// TIA Portal project "the last one" (V15)

(* hardware
DEVICE "S7-1200 station_1"  S7-1200 Station
   slot 0: "Rack_0"  S7-1200 Rack  Rack  V1.0
   slot 1: "PLC_1"  CPU 1212C AC/DC/Rly  6ES7 212-1BE40-0XB0  V4.0
   slot 101: "CM 1241 (RS422/485)_1"  6ES7 241-1CH32-0XB0  V2.2
DEVICE "S7-1200 station_3"  S7-1200 Station
   slot 0: "Rack_0"  S7-1200 Rack  Rack  V1.0
   slot 1: "PLC_3"  CPU 1212C AC/DC/Rly  6ES7 212-1BE31-0XB0  V3.0
*)

// ===== PLC "PLC_1"  CPU 1212C AC/DC/Rly =====

VAR_GLOBAL   // PLC tag table "Default tag table"
   "System_Byte" AT %MB1 : Byte;
   "FirstScan" AT %M1.0 : Bool;
   "DiagStatusUpdate" AT %M1.1 : Bool;
   "AlwaysTRUE" AT %M1.2 : Bool;
   "AlwaysFALSE" AT %M1.3 : Bool;
   "Clock_Byte" AT %MB0 : Byte;
   "Clock_10Hz" AT %M0.0 : Bool;
   "Clock_5Hz" AT %M0.1 : Bool;
   "Clock_2.5Hz" AT %M0.2 : Bool;
   "Clock_2Hz" AT %M0.3 : Bool;
   "Clock_1.25Hz" AT %M0.4 : Bool;
   "Clock_1Hz" AT %M0.5 : Bool;
   "Clock_0.625Hz" AT %M0.6 : Bool;
   "Clock_0.5Hz" AT %M0.7 : Bool;
   "Tag_1" AT %M2.0 : Bool;
   "Tag_2" AT %M2.1 : Bool;
   "Tag_3" AT %M2.2 : Bool;
   "Tag_4" AT %M2.3 : Bool;
   "Tag_5" AT %M2.4 : Bool;
   "Tag_6" AT %M2.5 : Bool;
   "freq" AT %MW10 : Word;
   "run" AT %MW12 : Word;
   "freq.refrance" AT %MW14 : Word;
   "volt" AT %MW16 : Word;
   "current" AT %MW18 : Word;
   "atomatic" AT %M2.6 : Bool;
   "manual" AT %M2.7 : Bool;
   "incoder_input" AT %ID1000 : DWord;
   "encoder" AT %MD40 : DInt;
   "panda(1)" AT %M3.0 : Bool;
   "start" AT %I0.1 : Bool;
   "reset" AT %I0.2 : Bool;
   "stop" AT %I0.3 : Bool;
   "stop_scada" AT %M3.1 : Bool;
   "reset_scada" AT %M3.2 : Bool;
   "start_scada" AT %M3.4 : Bool;
   "Tag_7" AT %M3.5 : Bool;
   "Tag_8" AT %M3.6 : Bool;
   "red" AT %MW20 : Word;
   "Tag_9" AT %MW22 : Int;
   "Tag_10" AT %M3.7 : Bool;
   "red valve" AT %Q0.0 : Bool;
   "Tag_11" AT %M4.0 : Bool;
   "Tag_12" AT %MW100 : Int;
   "Tag_13" AT %M4.1 : Bool;
   "Tag_14" AT %M4.2 : Bool;
   "reverse" AT %M4.3 : Bool;
   "Tag_15" AT %M4.4 : Bool;
   "Tag_16" AT %M4.5 : Bool;
   "Tag_17" AT %M4.6 : Bool;
   "Tag_18" AT %M4.7 : Bool;
   "green" AT %MW24 : Int;
   "Tag_19" AT %MW26 : Int;
   "green valve" AT %Q0.1 : Bool;
   "Tag_20" AT %M5.0 : Bool;
   "Tag_21" AT %M5.1 : Bool;
   "Tag_22" AT %M5.2 : Bool;
   "Tag_23" AT %M5.3 : Bool;
   "Tag_24" AT %M5.4 : Bool;
   "Tag_25" AT %M5.5 : Bool;
   "blue" AT %MW28 : Int;
   "Tag_27" AT %MW30 : Int;
   "blue valve" AT %Q0.2 : Bool;
   "Tag_28" AT %M5.6 : Bool;
   "Tag_26" AT %M5.7 : Bool;
   "Tag_29" AT %M6.0 : Bool;
   "Tag_30" AT %M6.1 : Bool;
   "Tag_31" AT %M6.2 : Bool;
   "Tag_32" AT %M6.3 : Bool;
   "Tag_33" AT %M6.4 : Bool;
   "Tag_34" AT %M6.5 : Bool;
   "Tag_35" AT %M6.6 : Bool;
   "Tag_36" AT %M6.7 : Bool;
   "cylinder" AT %Q0.3 : Bool;
   "Tag_37" AT %M7.0 : Bool;
   "mixer" AT %Q0.4 : Bool;
   "forward" AT %M7.1 : Bool;
   "Tag_38" AT %M7.2 : Bool;
   "Tag_39" AT %M7.3 : Bool;
   "Tag_40" AT %M7.5 : Bool;
   "Tag_41" AT %M7.6 : Bool;
   "Tag_42" AT %M7.7 : Bool;
   "Tag_43" AT %M8.0 : Bool;
   "Tag_44" AT %M8.1 : Bool;
   "Tag_45" AT %M8.2 : Bool;
   "m_redvalve" AT %M8.3 : Bool;
   "m_greenvalve" AT %M8.4 : Bool;
   "Tag_48" AT %M8.5 : Bool;
   "m_bluevalve" AT %M8.6 : Bool;
   "m_forward" AT %M8.7 : Bool;
   "m_reverse" AT %M9.0 : Bool;
   "Tag_52" AT %M9.1 : Bool;
   "Tag_46" AT %M9.2 : Bool;
   "Tag_47" AT %M9.3 : Bool;
   "Tag_49" AT %M9.4 : Bool;
   "Tag_50" AT %M34.0 : Bool;
   "Tag_51" AT %M90.0 : Bool;
   "Tag_53" AT %MW102 : Int;
   "Tag_54" AT %MW104 : Int;
   "Tag_55" AT %M90.1 : Bool;
   "Tag_56" AT %MD50 : DWord;
   "Tag_57" AT %MD54 : DWord;
   "Tag_58" AT %M50.0 : Bool;
   "Tag_59" AT %M50.1 : Bool;
   "n0" AT %M58.0 : Bool;
   "n1" AT %M58.1 : Bool;
   "n2" AT %M58.2 : Bool;
   "n3" AT %M58.3 : Bool;
   "n4" AT %M58.4 : Bool;
   "n5" AT %M58.5 : Bool;
   "n6" AT %M58.6 : Bool;
   "n7" AT %M58.7 : Bool;
   "p0" AT %M59.0 : Bool;
   "p1" AT %M59.1 : Bool;
   "p2" AT %M59.2 : Bool;
   "p3" AT %M59.3 : Bool;
   "p4" AT %M59.4 : Bool;
   "p5" AT %M59.5 : Bool;
   "p6" AT %M59.6 : Bool;
   "p7" AT %M59.7 : Bool;
   "p8" AT %M60.0 : Bool;
   "p9" AT %M60.1 : Bool;
   "X" AT %M110.0 : Bool;
   "Tag_60" AT %MW60 : Int;
   "r0" AT %M62.0 : Bool;
   "r1" AT %M62.1 : Bool;
   "r2" AT %M62.2 : Bool;
   "r3" AT %M62.3 : Bool;
   "r4" AT %M62.4 : Bool;
   "r5" AT %M62.5 : Bool;
   "r6" AT %M62.6 : Bool;
   "r7" AT %M62.7 : Bool;
   "r8" AT %M63.0 : Bool;
   "r9" AT %M63.1 : Bool;
   "t1" AT %M63.2 : Bool;
   "t2" AT %M63.3 : Bool;
   "t3" AT %M63.4 : Bool;
   "t4" AT %M63.5 : Bool;
   "t5" AT %M63.6 : Bool;
   "t6" AT %M63.7 : Bool;
   "t7" AT %M64.0 : Bool;
   "t8" AT %M64.1 : Bool;
   "Tag_61" AT %MW80 : Int;
   "Tag_62" AT %MW120 : Word;
   "Tag_63" AT %MW90 : Int;
   "Tag_64" AT %MW40 : Word;
   "Tag_65" AT %MW82 : Int;
   "Tag_66" AT %MW122 : Word;
   "Tag_67" AT %MW92 : Int;
   "Tag_68" AT %MW124 : Word;
   "Tag_69" AT %MW94 : Int;
   "Tag_70" AT %MW84 : Int;
   "Tag_71" AT %MW130 : Int;
   "Tag_72" AT %MW132 : Int;
   "Tag_73" AT %MW134 : Int;
   "Tag_74" AT %MW136 : Int;
   "p11" AT %M138.0 : Bool;
   "p12" AT %M138.1 : Bool;
   "p13" AT %M138.2 : Bool;
   "p14" AT %M138.3 : Bool;
   "Tag_75" AT %MW50 : Word;
   "rstop" AT %M138.4 : Bool;
   "Tag_76" AT %MW86 : Word;
   "Tag_77" AT %M87.0 : Bool;
   "Tag_78" AT %M87.1 : Bool;
   "Tag_79" AT %M87.5 : Bool;
   "Tag_80" AT %M150.0 : Bool;
   "Tag_81" AT %M150.2 : Bool;
   "Tag_82" AT %M150.3 : Bool;
   "Tag_83" AT %M150.4 : Bool;
   "Tag_84" AT %M150.5 : Bool;
   "Tag_85" AT %M150.6 : Bool;
   "Tag_86" AT %M151.0 : Bool;
   "Tag_87" AT %M151.2 : Bool;
   "Tag_88" AT %M153.0 : Bool;
   "valve 1" AT %M160.0 : Bool;
   "valve 2" AT %M160.1 : Bool;
   "valve 3" AT %M160.2 : Bool;
   "cylinder_scada" AT %M160.3 : Bool;
   "mixer_scada" AT %M160.4 : Bool;
   "forward_scada" AT %M160.5 : Bool;
   "reverse_scada" AT %M160.6 : Bool;
   "Tag_89" AT %M166.0 : Bool;
   "Tag_90" AT %M166.1 : Bool;
   "Tag_91" AT %M166.2 : Bool;
   "Tag_92" AT %M166.3 : Bool;
   "Tag_93" AT %M170.0 : Bool;
   "Tag_94" AT %M171.0 : Bool;
   "Tag_95" AT %M170.1 : Bool;
   "Tag_96" AT %M171.1 : Bool;
   "Tag_97" AT %M170.3 : Bool;
   "Tag_98" AT %M171.3 : Bool;
   "Tag_99" AT %M170.2 : Bool;
   "Tag_100" AT %M171.2 : Bool;
END_VAR

DATA_BLOCK "auto_DB"   // DB11
{ S7_Optimized_Access := 'TRUE' }
VERSION : 0.1
// stored: InstanceOfName auto
"auto"
BEGIN
END_DATA_BLOCK

// folder: System blocks/Program resources

DATA_BLOCK "IEC_Counter_0_DB"   // DB4
{ S7_Optimized_Access := 'TRUE' }
AUTHOR : Simatic
FAMILY : IEC
NAME : CNTR
VERSION : 1.0
// stored: InstanceOfName IEC_COUNTER
"IEC_COUNTER"
BEGIN
END_DATA_BLOCK

DATA_BLOCK "IEC_Timer_0_DB"   // DB5
{ S7_Optimized_Access := 'TRUE' }
AUTHOR : Simatic
FAMILY : IEC
NAME : IEC_TMR
VERSION : 1.0
// stored: InstanceOfName IEC_TIMER
"IEC_TIMER"
BEGIN
END_DATA_BLOCK

DATA_BLOCK "IEC_Timer_0_DB_1"   // DB6
{ S7_Optimized_Access := 'TRUE' }
AUTHOR : Simatic
FAMILY : IEC
NAME : IEC_TMR
VERSION : 1.0
// stored: InstanceOfName IEC_TIMER
"IEC_TIMER"
BEGIN
END_DATA_BLOCK

DATA_BLOCK "IEC_Timer_0_DB_2"   // DB7
{ S7_Optimized_Access := 'TRUE' }
AUTHOR : Simatic
FAMILY : IEC
NAME : IEC_TMR
VERSION : 1.0
// stored: InstanceOfName IEC_TIMER
"IEC_TIMER"
BEGIN
END_DATA_BLOCK

DATA_BLOCK "IEC_Timer_0_DB_3"   // DB8
{ S7_Optimized_Access := 'TRUE' }
AUTHOR : Simatic
FAMILY : IEC
NAME : IEC_TMR
VERSION : 1.0
// stored: InstanceOfName IEC_TIMER
"IEC_TIMER"
BEGIN
END_DATA_BLOCK

DATA_BLOCK "IEC_Counter_0_DB_1"   // DB9
{ S7_Optimized_Access := 'TRUE' }
AUTHOR : Simatic
FAMILY : IEC
NAME : CNTR
VERSION : 1.0
// stored: InstanceOfName IEC_COUNTER
"IEC_COUNTER"
BEGIN
END_DATA_BLOCK

DATA_BLOCK "IEC_Timer_0_DB_4"   // DB10
{ S7_Optimized_Access := 'TRUE' }
AUTHOR : Simatic
FAMILY : IEC
NAME : IEC_TMR
VERSION : 1.0
// stored: InstanceOfName IEC_TIMER
"IEC_TIMER"
BEGIN
END_DATA_BLOCK

DATA_BLOCK "IEC_Counter_0_DB_2"   // DB13
{ S7_Optimized_Access := 'TRUE' }
AUTHOR : Simatic
FAMILY : IEC
NAME : CNTR
VERSION : 1.0
// stored: InstanceOfName IEC_COUNTER
"IEC_COUNTER"
BEGIN
END_DATA_BLOCK

DATA_BLOCK "IEC_Counter_0_DB_3"   // DB14
{ S7_Optimized_Access := 'TRUE' }
AUTHOR : Simatic
FAMILY : IEC
NAME : CNTR
VERSION : 1.0
// stored: InstanceOfName IEC_COUNTER
"IEC_COUNTER"
BEGIN
END_DATA_BLOCK

// folder: (top level)

FUNCTION_BLOCK "auto"   // FB1, LAD
{ S7_Optimized_Access := 'TRUE' }
VERSION : 0.1
   VAR_TEMP   // added for the SCL form of the ladder/FBD networks
      _w1 : Bool;
      _w2 : Bool;
      _w3 : Bool;
      _w4 : Bool;
   END_VAR
BEGIN

REGION Network 1
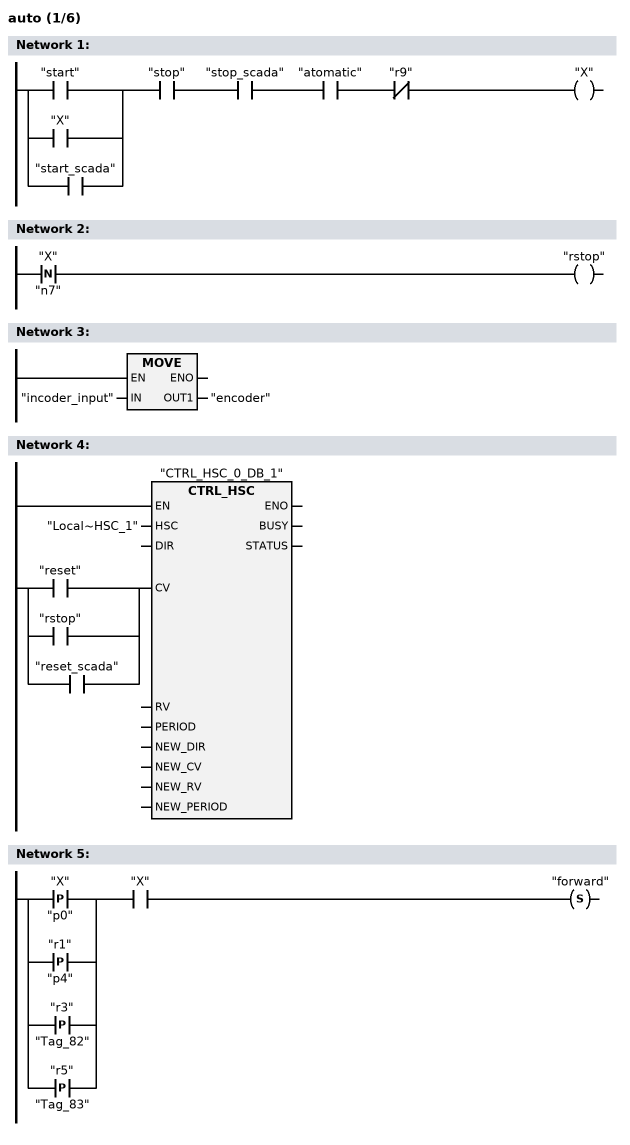
   RUNG wire#powerrail
      Contact( "start" )
      wire#w1
      Contact( "stop" )
      Contact( "stop_scada" )
      Contact( "atomatic" )
      I_Contact( "r9" )
      Coil( "X" )
   END_RUNG
   RUNG wire#powerrail
      Contact( "X" )
   END_RUNG wire#w1
   RUNG wire#powerrail
      Contact( "start_scada" )
   END_RUNG wire#w1
   // the same network as SCL:
   "X" := ("start" OR "X" OR "start_scada") AND "stop" AND "stop_scada" AND "atomatic" AND NOT "r9";
END_REGION

REGION Network 2
   RUNG wire#powerrail
      N_Contact(operand := "X", bit := "n7")
      Coil( "rstop" )
   END_RUNG
   // the same network as SCL:
   #_w1 := NOT "X" AND "n7";   // falling edge of "X"
   "n7" := "X";
   "rstop" := #_w1;
END_REGION

REGION Network 3
   RUNG wire#powerrail
      Move(in := "incoder_input", out1 => "encoder")
   END_RUNG
   // the same network as SCL:
   "encoder" := "incoder_input";
END_REGION

REGION Network 4
   "CTRL_HSC_0_DB_1"(HSC := "Local~HSC_1", CV := "reset" OR "rstop" OR "reset_scada");   // CTRL_HSC
END_REGION

REGION Network 5
   RUNG wire#powerrail
      P_Contact(operand := "X", bit := "p0")
      wire#w1
      Contact( "X" )
      S_Coil( "forward" )
   END_RUNG
   RUNG wire#powerrail
      P_Contact(operand := "r1", bit := "p4")
   END_RUNG wire#w1
   RUNG wire#powerrail
      P_Contact(operand := "r3", bit := "Tag_82")
   END_RUNG wire#w1
   RUNG wire#powerrail
      P_Contact(operand := "r5", bit := "Tag_83")
   END_RUNG wire#w1
   // the same network as SCL:
   #_w1 := "X" AND NOT "p0";   // rising edge of "X"
   "p0" := "X";
   #_w2 := "r1" AND NOT "p4";   // rising edge of "r1"
   "p4" := "r1";
   #_w3 := "r3" AND NOT "Tag_82";   // rising edge of "r3"
   "Tag_82" := "r3";
   #_w4 := "r5" AND NOT "Tag_83";   // rising edge of "r5"
   "Tag_83" := "r5";
   IF (#_w1 OR #_w2 OR #_w3 OR #_w4) AND "X" THEN "forward" := TRUE; END_IF;
END_REGION

REGION Network 6
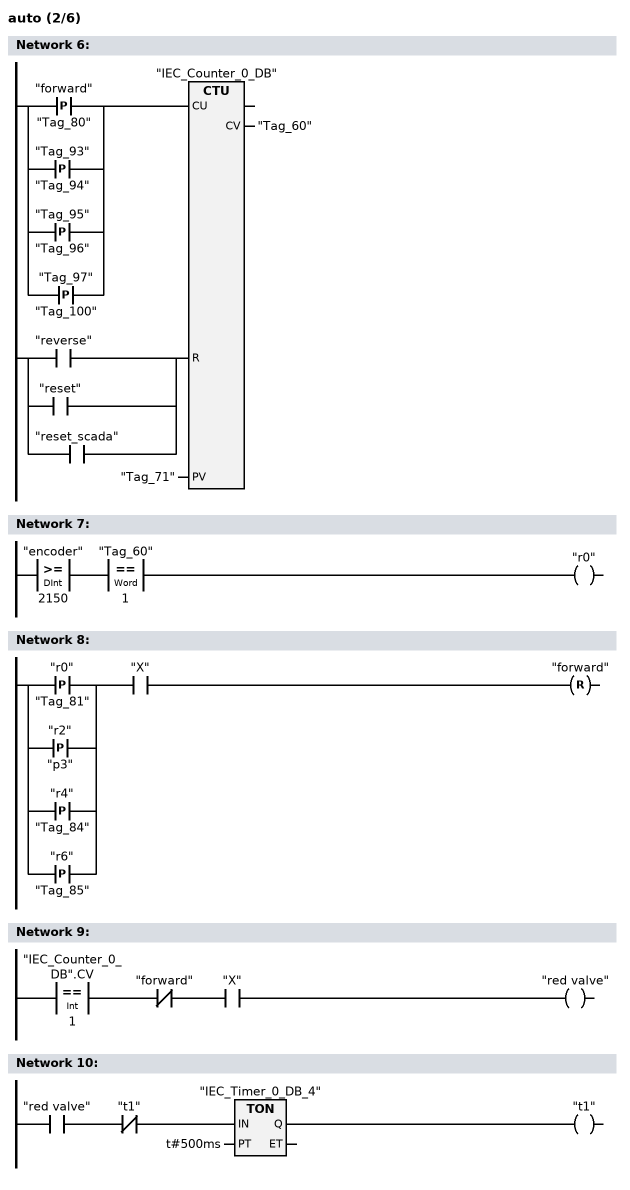
   #_w1 := "forward" AND NOT "Tag_80";   // rising edge of "forward"
   "Tag_80" := "forward";
   #_w2 := "Tag_93" AND NOT "Tag_94";   // rising edge of "Tag_93"
   "Tag_94" := "Tag_93";
   #_w3 := "Tag_95" AND NOT "Tag_96";   // rising edge of "Tag_95"
   "Tag_96" := "Tag_95";
   #_w4 := "Tag_97" AND NOT "Tag_100";   // rising edge of "Tag_97"
   "Tag_100" := "Tag_97";
   "IEC_Counter_0_DB".CTU(CU := #_w1 OR #_w2 OR #_w3 OR #_w4,
                          R := "reverse" OR "reset" OR "reset_scada",
                          PV := "Tag_71",
                          CV => "Tag_60");
END_REGION

REGION Network 7
   RUNG wire#powerrail
      { S7_Templates := "SrcType := DInt" } GE_Contact(in1 := "encoder", in2 := 2150)
      { S7_Templates := "SrcType := Word" } EQ_Contact(in1 := "Tag_60", in2 := 1)
      Coil( "r0" )
   END_RUNG
   // the same network as SCL:
   "r0" := ("encoder" >= 2150) AND ("Tag_60" = 1);
END_REGION

REGION Network 8
   RUNG wire#powerrail
      P_Contact(operand := "r0", bit := "Tag_81")
      wire#w1
      Contact( "X" )
      R_Coil( "forward" )
   END_RUNG
   RUNG wire#powerrail
      P_Contact(operand := "r2", bit := "p3")
   END_RUNG wire#w1
   RUNG wire#powerrail
      P_Contact(operand := "r4", bit := "Tag_84")
   END_RUNG wire#w1
   RUNG wire#powerrail
      P_Contact(operand := "r6", bit := "Tag_85")
   END_RUNG wire#w1
   // the same network as SCL:
   #_w1 := "r0" AND NOT "Tag_81";   // rising edge of "r0"
   "Tag_81" := "r0";
   #_w2 := "r2" AND NOT "p3";   // rising edge of "r2"
   "p3" := "r2";
   #_w3 := "r4" AND NOT "Tag_84";   // rising edge of "r4"
   "Tag_84" := "r4";
   #_w4 := "r6" AND NOT "Tag_85";   // rising edge of "r6"
   "Tag_85" := "r6";
   IF (#_w1 OR #_w2 OR #_w3 OR #_w4) AND "X" THEN "forward" := FALSE; END_IF;
END_REGION

REGION Network 9
   RUNG wire#powerrail
      { S7_Templates := "SrcType := Int" } EQ_Contact(in1 := "IEC_Counter_0_DB".CV, in2 := 1)
      I_Contact( "forward" )
      Contact( "X" )
      Coil( "red valve" )
   END_RUNG
   // the same network as SCL:
   "red valve" := ("IEC_Counter_0_DB".CV = 1) AND NOT "forward" AND "X";
END_REGION

REGION Network 10
   "IEC_Timer_0_DB_4".TON(IN := "red valve" AND NOT "t1", PT := t#500ms);
   "t1" := "IEC_Timer_0_DB_4".Q;
END_REGION

REGION Network 11
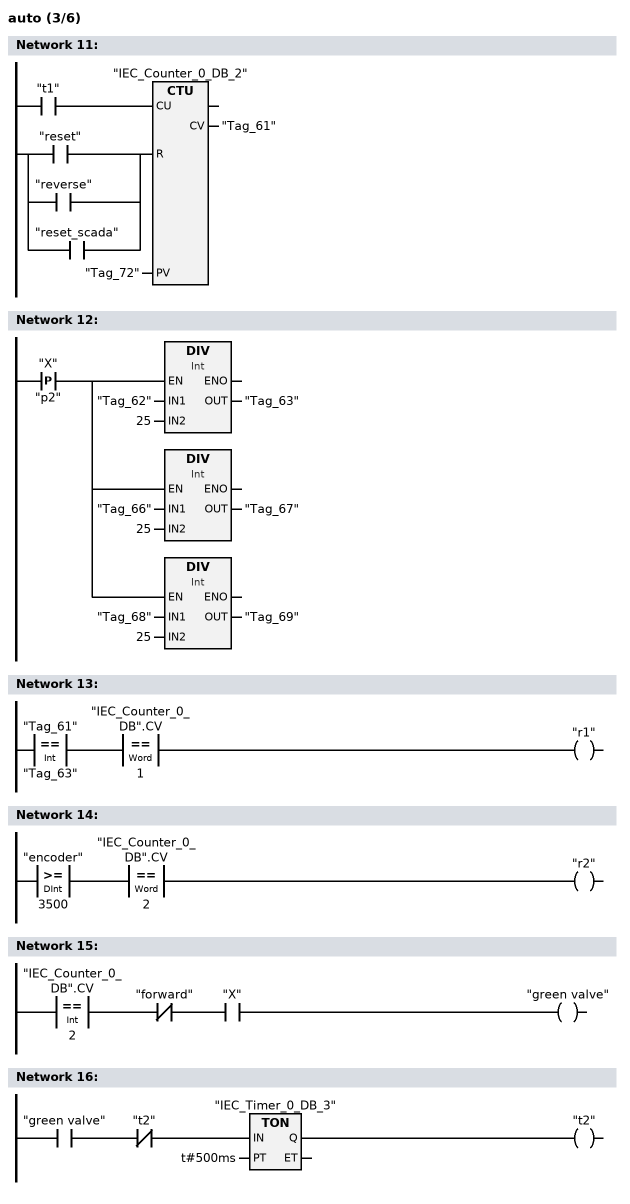
   "IEC_Counter_0_DB_2".CTU(CU := "t1",
                           R := "reset" OR "reverse" OR "reset_scada",
                           PV := "Tag_72",
                           CV => "Tag_61");
END_REGION

REGION Network 12
   RUNG wire#powerrail
      P_Contact(operand := "X", bit := "p2")
      wire#w1
      { S7_Templates := "SrcType := Int" } Div(in1 := "Tag_62", in2 := 25, out => "Tag_63")
   END_RUNG
   RUNG wire#w1
      { S7_Templates := "SrcType := Int" } Div(in1 := "Tag_66", in2 := 25, out => "Tag_67")
   END_RUNG
   RUNG wire#w1
      { S7_Templates := "SrcType := Int" } Div(in1 := "Tag_68", in2 := 25, out => "Tag_69")
   END_RUNG
   // the same network as SCL:
   #_w1 := "X" AND NOT "p2";   // rising edge of "X"
   "p2" := "X";
   IF #_w1 THEN
       "Tag_63" := "Tag_62" / 25;
       "Tag_67" := "Tag_66" / 25;
       "Tag_69" := "Tag_68" / 25;
   END_IF;
END_REGION

REGION Network 13
   RUNG wire#powerrail
      { S7_Templates := "SrcType := Int" } EQ_Contact(in1 := "Tag_61", in2 := "Tag_63")
      { S7_Templates := "SrcType := Word" } EQ_Contact(in1 := "IEC_Counter_0_DB".CV, in2 := 1)
      Coil( "r1" )
   END_RUNG
   // the same network as SCL:
   "r1" := ("Tag_61" = "Tag_63") AND ("IEC_Counter_0_DB".CV = 1);
END_REGION

REGION Network 14
   RUNG wire#powerrail
      { S7_Templates := "SrcType := DInt" } GE_Contact(in1 := "encoder", in2 := 3500)
      { S7_Templates := "SrcType := Word" } EQ_Contact(in1 := "IEC_Counter_0_DB".CV, in2 := 2)
      Coil( "r2" )
   END_RUNG
   // the same network as SCL:
   "r2" := ("encoder" >= 3500) AND ("IEC_Counter_0_DB".CV = 2);
END_REGION

REGION Network 15
   RUNG wire#powerrail
      { S7_Templates := "SrcType := Int" } EQ_Contact(in1 := "IEC_Counter_0_DB".CV, in2 := 2)
      I_Contact( "forward" )
      Contact( "X" )
      Coil( "green valve" )
   END_RUNG
   // the same network as SCL:
   "green valve" := ("IEC_Counter_0_DB".CV = 2) AND NOT "forward" AND "X";
END_REGION

REGION Network 16
   "IEC_Timer_0_DB_3".TON(IN := "green valve" AND NOT "t2", PT := t#500ms);
   "t2" := "IEC_Timer_0_DB_3".Q;
END_REGION

REGION Network 17
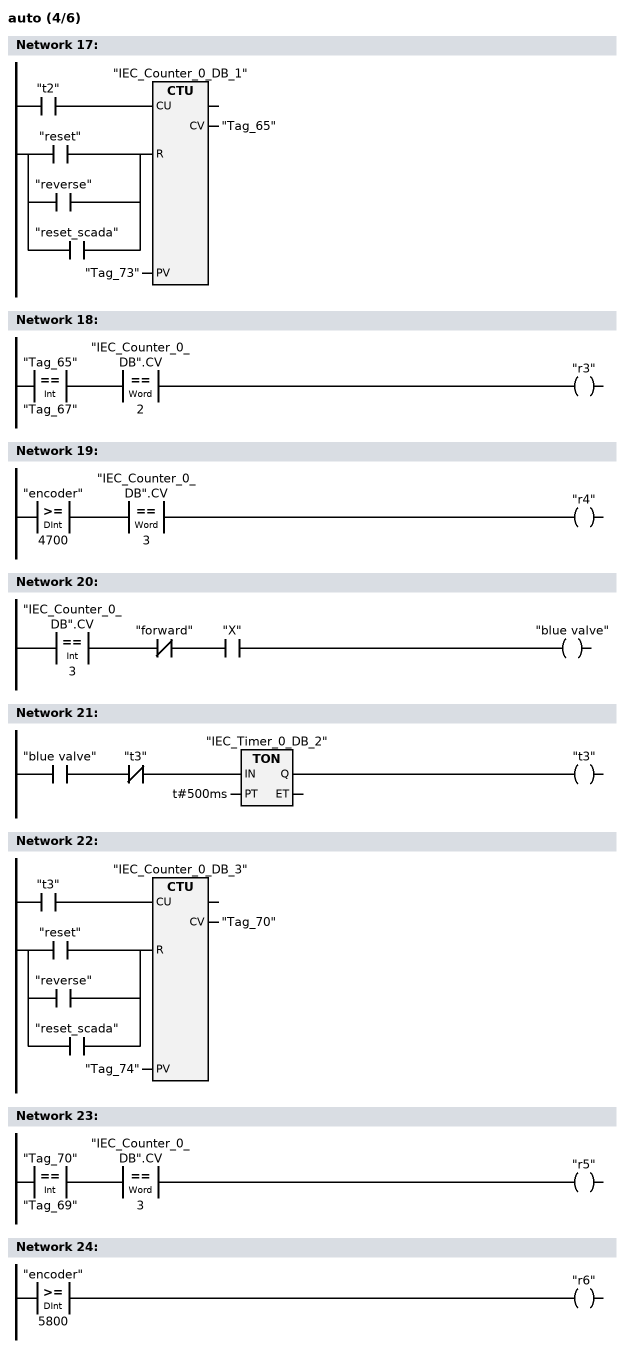
   "IEC_Counter_0_DB_1".CTU(CU := "t2",
                           R := "reset" OR "reverse" OR "reset_scada",
                           PV := "Tag_73",
                           CV => "Tag_65");
END_REGION

REGION Network 18
   RUNG wire#powerrail
      { S7_Templates := "SrcType := Int" } EQ_Contact(in1 := "Tag_65", in2 := "Tag_67")
      { S7_Templates := "SrcType := Word" } EQ_Contact(in1 := "IEC_Counter_0_DB".CV, in2 := 2)
      Coil( "r3" )
   END_RUNG
   // the same network as SCL:
   "r3" := ("Tag_65" = "Tag_67") AND ("IEC_Counter_0_DB".CV = 2);
END_REGION

REGION Network 19
   RUNG wire#powerrail
      { S7_Templates := "SrcType := DInt" } GE_Contact(in1 := "encoder", in2 := 4700)
      { S7_Templates := "SrcType := Word" } EQ_Contact(in1 := "IEC_Counter_0_DB".CV, in2 := 3)
      Coil( "r4" )
   END_RUNG
   // the same network as SCL:
   "r4" := ("encoder" >= 4700) AND ("IEC_Counter_0_DB".CV = 3);
END_REGION

REGION Network 20
   RUNG wire#powerrail
      { S7_Templates := "SrcType := Int" } EQ_Contact(in1 := "IEC_Counter_0_DB".CV, in2 := 3)
      I_Contact( "forward" )
      Contact( "X" )
      Coil( "blue valve" )
   END_RUNG
   // the same network as SCL:
   "blue valve" := ("IEC_Counter_0_DB".CV = 3) AND NOT "forward" AND "X";
END_REGION

REGION Network 21
   "IEC_Timer_0_DB_2".TON(IN := "blue valve" AND NOT "t3", PT := t#500ms);
   "t3" := "IEC_Timer_0_DB_2".Q;
END_REGION

REGION Network 22
   "IEC_Counter_0_DB_3".CTU(CU := "t3",
                           R := "reset" OR "reverse" OR "reset_scada",
                           PV := "Tag_74",
                           CV => "Tag_70");
END_REGION

REGION Network 23
   RUNG wire#powerrail
      { S7_Templates := "SrcType := Int" } EQ_Contact(in1 := "Tag_70", in2 := "Tag_69")
      { S7_Templates := "SrcType := Word" } EQ_Contact(in1 := "IEC_Counter_0_DB".CV, in2 := 3)
      Coil( "r5" )
   END_RUNG
   // the same network as SCL:
   "r5" := ("Tag_70" = "Tag_69") AND ("IEC_Counter_0_DB".CV = 3);
END_REGION

REGION Network 24
   RUNG wire#powerrail
      { S7_Templates := "SrcType := DInt" } GE_Contact(in1 := "encoder", in2 := 5800)
      Coil( "r6" )
   END_RUNG
   // the same network as SCL:
   "r6" := "encoder" >= 5800;
END_REGION

REGION Network 25
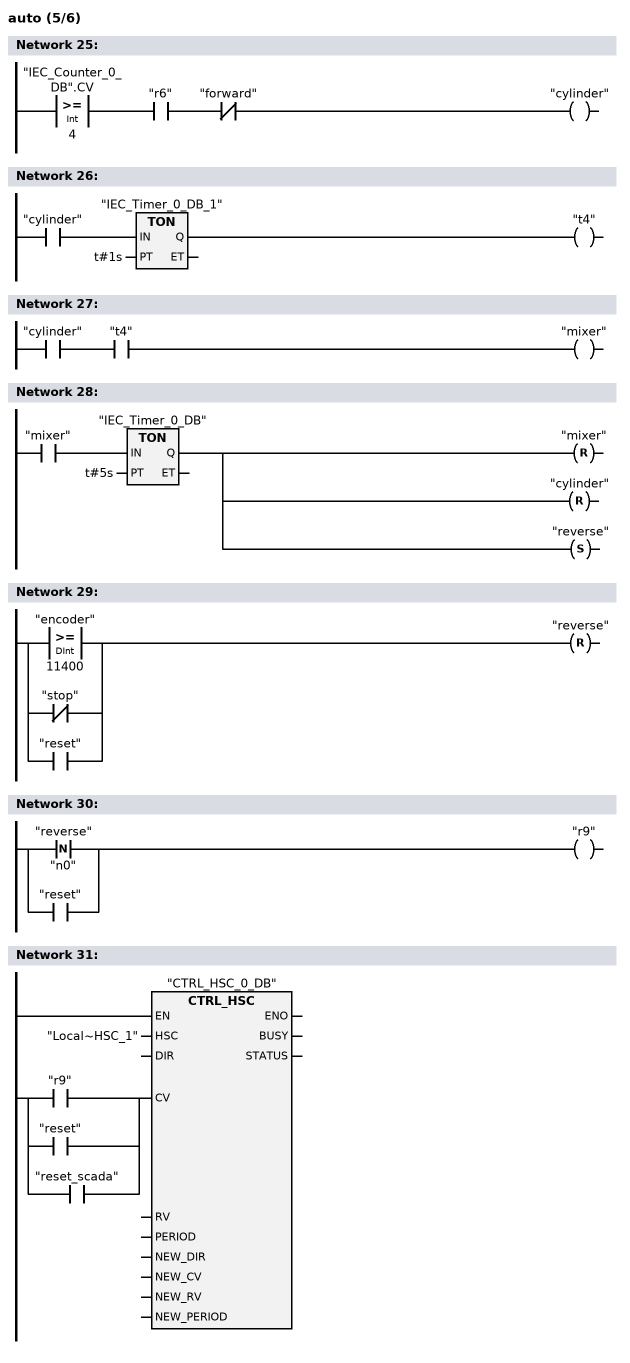
   RUNG wire#powerrail
      { S7_Templates := "SrcType := Int" } GE_Contact(in1 := "IEC_Counter_0_DB".CV, in2 := 4)
      Contact( "r6" )
      I_Contact( "forward" )
      Coil( "cylinder" )
   END_RUNG
   // the same network as SCL:
   "cylinder" := ("IEC_Counter_0_DB".CV >= 4) AND "r6" AND NOT "forward";
END_REGION

REGION Network 26
   "IEC_Timer_0_DB_1".TON(IN := "cylinder", PT := t#1s);
   "t4" := "IEC_Timer_0_DB_1".Q;
END_REGION

REGION Network 27
   RUNG wire#powerrail
      Contact( "cylinder" )
      Contact( "t4" )
      Coil( "mixer" )
   END_RUNG
   // the same network as SCL:
   "mixer" := "cylinder" AND "t4";
END_REGION

REGION Network 28
   "IEC_Timer_0_DB".TON(IN := "mixer", PT := t#5s);
   IF "IEC_Timer_0_DB".Q THEN
       "mixer" := FALSE;
       "cylinder" := FALSE;
       "reverse" := TRUE;
   END_IF;
END_REGION

REGION Network 29
   RUNG wire#powerrail
      { S7_Templates := "SrcType := DInt" } GE_Contact(in1 := "encoder", in2 := 11400)
      wire#w1
      R_Coil( "reverse" )
   END_RUNG
   RUNG wire#powerrail
      I_Contact( "stop" )
   END_RUNG wire#w1
   RUNG wire#powerrail
      Contact( "reset" )
   END_RUNG wire#w1
   // the same network as SCL:
   IF ("encoder" >= 11400) OR NOT "stop" OR "reset" THEN "reverse" := FALSE; END_IF;
END_REGION

REGION Network 30
   RUNG wire#powerrail
      N_Contact(operand := "reverse", bit := "n0")
      wire#w1
      Coil( "r9" )
   END_RUNG
   RUNG wire#powerrail
      Contact( "reset" )
   END_RUNG wire#w1
   // the same network as SCL:
   #_w1 := NOT "reverse" AND "n0";   // falling edge of "reverse"
   "n0" := "reverse";
   "r9" := #_w1 OR "reset";
END_REGION

REGION Network 31
   "CTRL_HSC_0_DB"(HSC := "Local~HSC_1", CV := "r9" OR "reset" OR "reset_scada");   // CTRL_HSC
END_REGION

REGION Network 32
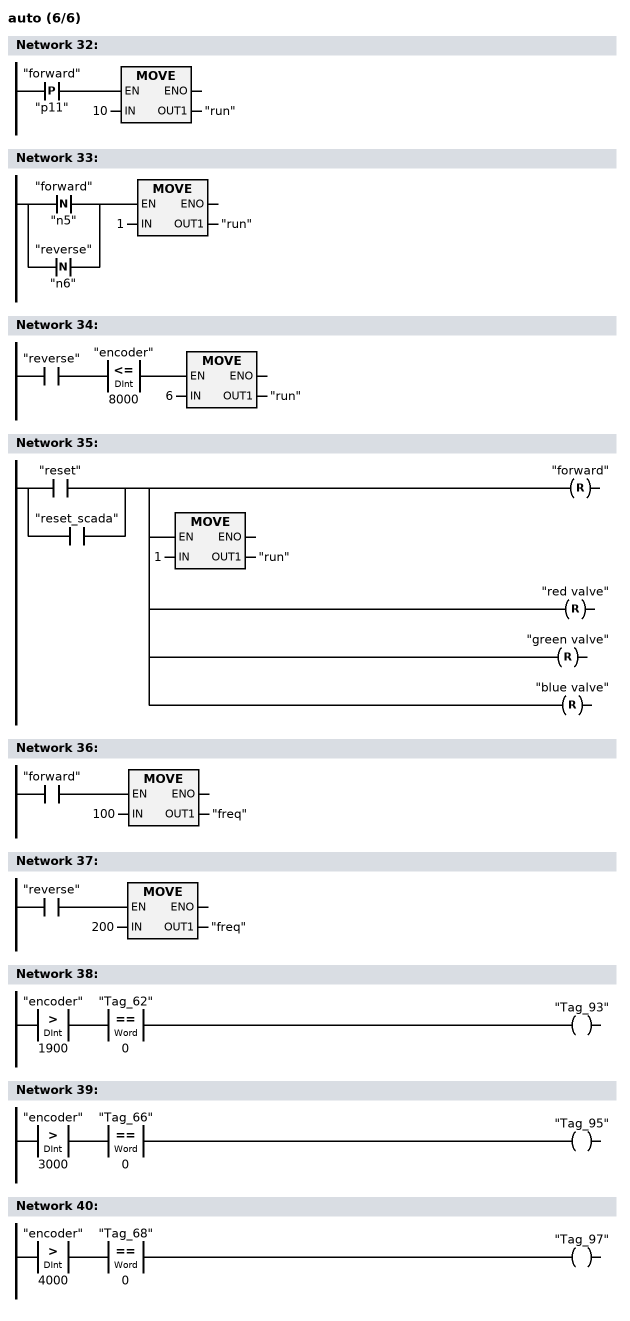
   RUNG wire#powerrail
      P_Contact(operand := "forward", bit := "p11")
      Move(in := 10, out1 => "run")
   END_RUNG
   // the same network as SCL:
   #_w1 := "forward" AND NOT "p11";   // rising edge of "forward"
   "p11" := "forward";
   IF #_w1 THEN "run" := 10; END_IF;
END_REGION

REGION Network 33
   RUNG wire#powerrail
      N_Contact(operand := "forward", bit := "n5")
      wire#w1
      Move(in := 1, out1 => "run")
   END_RUNG
   RUNG wire#powerrail
      N_Contact(operand := "reverse", bit := "n6")
   END_RUNG wire#w1
   // the same network as SCL:
   #_w1 := NOT "forward" AND "n5";   // falling edge of "forward"
   "n5" := "forward";
   #_w2 := NOT "reverse" AND "n6";   // falling edge of "reverse"
   "n6" := "reverse";
   IF #_w1 OR #_w2 THEN "run" := 1; END_IF;
END_REGION

REGION Network 34
   RUNG wire#powerrail
      Contact( "reverse" )
      { S7_Templates := "SrcType := DInt" } LE_Contact(in1 := "encoder", in2 := 8000)
      Move(in := 6, out1 => "run")
   END_RUNG
   // the same network as SCL:
   IF "reverse" AND ("encoder" <= 8000) THEN "run" := 6; END_IF;
END_REGION

REGION Network 35
   RUNG wire#powerrail
      Contact( "reset" )
      wire#w1
      R_Coil( "forward" )
   END_RUNG
   RUNG wire#powerrail
      Contact( "reset_scada" )
   END_RUNG wire#w1
   RUNG wire#w1
      Move(in := 1, out1 => "run")
   END_RUNG
   RUNG wire#w1
      R_Coil( "red valve" )
   END_RUNG
   RUNG wire#w1
      R_Coil( "green valve" )
   END_RUNG
   RUNG wire#w1
      R_Coil( "blue valve" )
   END_RUNG
   // the same network as SCL:
   IF "reset" OR "reset_scada" THEN
       "forward" := FALSE;
       "run" := 1;
       "red valve" := FALSE;
       "green valve" := FALSE;
       "blue valve" := FALSE;
   END_IF;
END_REGION

REGION Network 36
   RUNG wire#powerrail
      Contact( "forward" )
      Move(in := 100, out1 => "freq")
   END_RUNG
   // the same network as SCL:
   IF "forward" THEN "freq" := 100; END_IF;
END_REGION

REGION Network 37
   RUNG wire#powerrail
      Contact( "reverse" )
      Move(in := 200, out1 => "freq")
   END_RUNG
   // the same network as SCL:
   IF "reverse" THEN "freq" := 200; END_IF;
END_REGION

REGION Network 38
   RUNG wire#powerrail
      { S7_Templates := "SrcType := DInt" } GT_Contact(in1 := "encoder", in2 := 1900)
      { S7_Templates := "SrcType := Word" } EQ_Contact(in1 := "Tag_62", in2 := 0)
      Coil( "Tag_93" )
   END_RUNG
   // the same network as SCL:
   "Tag_93" := ("encoder" > 1900) AND ("Tag_62" = 0);
END_REGION

REGION Network 39
   RUNG wire#powerrail
      { S7_Templates := "SrcType := DInt" } GT_Contact(in1 := "encoder", in2 := 3000)
      { S7_Templates := "SrcType := Word" } EQ_Contact(in1 := "Tag_66", in2 := 0)
      Coil( "Tag_95" )
   END_RUNG
   // the same network as SCL:
   "Tag_95" := ("encoder" > 3000) AND ("Tag_66" = 0);
END_REGION

REGION Network 40
   RUNG wire#powerrail
      { S7_Templates := "SrcType := DInt" } GT_Contact(in1 := "encoder", in2 := 4000)
      { S7_Templates := "SrcType := Word" } EQ_Contact(in1 := "Tag_68", in2 := 0)
      Coil( "Tag_97" )
   END_RUNG
   // the same network as SCL:
   "Tag_97" := ("encoder" > 4000) AND ("Tag_68" = 0);
END_REGION
END_FUNCTION_BLOCK

FUNCTION "manu" : Void   // FC1, LAD
{ S7_Optimized_Access := 'TRUE' }
VERSION : 0.1
   VAR_TEMP   // added for the SCL form of the ladder/FBD networks
      _w1 : Bool;
      _w2 : Bool;
   END_VAR
BEGIN

REGION Network 1
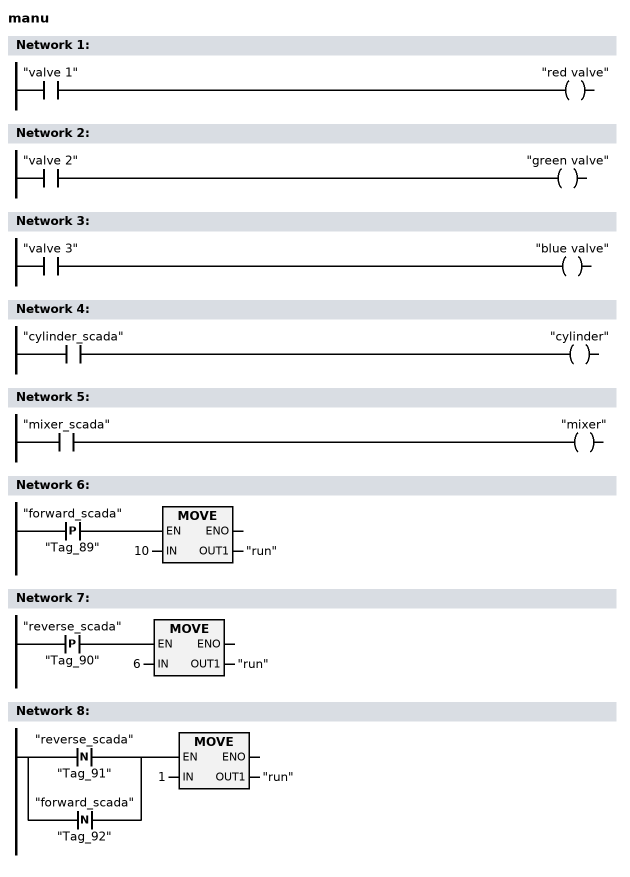
   RUNG wire#powerrail
      Contact( "valve 1" )
      Coil( "red valve" )
   END_RUNG
   // the same network as SCL:
   "red valve" := "valve 1";
END_REGION

REGION Network 2
   RUNG wire#powerrail
      Contact( "valve 2" )
      Coil( "green valve" )
   END_RUNG
   // the same network as SCL:
   "green valve" := "valve 2";
END_REGION

REGION Network 3
   RUNG wire#powerrail
      Contact( "valve 3" )
      Coil( "blue valve" )
   END_RUNG
   // the same network as SCL:
   "blue valve" := "valve 3";
END_REGION

REGION Network 4
   RUNG wire#powerrail
      Contact( "cylinder_scada" )
      Coil( "cylinder" )
   END_RUNG
   // the same network as SCL:
   "cylinder" := "cylinder_scada";
END_REGION

REGION Network 5
   RUNG wire#powerrail
      Contact( "mixer_scada" )
      Coil( "mixer" )
   END_RUNG
   // the same network as SCL:
   "mixer" := "mixer_scada";
END_REGION

REGION Network 6
   RUNG wire#powerrail
      P_Contact(operand := "forward_scada", bit := "Tag_89")
      Move(in := 10, out1 => "run")
   END_RUNG
   // the same network as SCL:
   #_w1 := "forward_scada" AND NOT "Tag_89";   // rising edge of "forward_scada"
   "Tag_89" := "forward_scada";
   IF #_w1 THEN "run" := 10; END_IF;
END_REGION

REGION Network 7
   RUNG wire#powerrail
      P_Contact(operand := "reverse_scada", bit := "Tag_90")
      Move(in := 6, out1 => "run")
   END_RUNG
   // the same network as SCL:
   #_w1 := "reverse_scada" AND NOT "Tag_90";   // rising edge of "reverse_scada"
   "Tag_90" := "reverse_scada";
   IF #_w1 THEN "run" := 6; END_IF;
END_REGION

REGION Network 8
   RUNG wire#powerrail
      N_Contact(operand := "reverse_scada", bit := "Tag_91")
      wire#w1
      Move(in := 1, out1 => "run")
   END_RUNG
   RUNG wire#powerrail
      N_Contact(operand := "forward_scada", bit := "Tag_92")
   END_RUNG wire#w1
   // the same network as SCL:
   #_w1 := NOT "reverse_scada" AND "Tag_91";   // falling edge of "reverse_scada"
   "Tag_91" := "reverse_scada";
   #_w2 := NOT "forward_scada" AND "Tag_92";   // falling edge of "forward_scada"
   "Tag_92" := "forward_scada";
   IF #_w1 OR #_w2 THEN "run" := 1; END_IF;
END_REGION
END_FUNCTION

ORGANIZATION_BLOCK "Main"   // OB1, LAD, ProgramCycle
TITLE = "Main Program Sweep (Cycle)"
{ S7_Optimized_Access := 'TRUE' }
VERSION : 0.1
   VAR_INPUT
      Initial_Call : Bool;   // Initial call of this OB
      Remanence : Bool;   // =True, if remanent data are available
   END_VAR
   VAR_TEMP   // added for the SCL form of the ladder/FBD networks
      _w1 : Bool;
      _w2 : Bool;
      _w3 : Bool;
   END_VAR
BEGIN

REGION Network 1
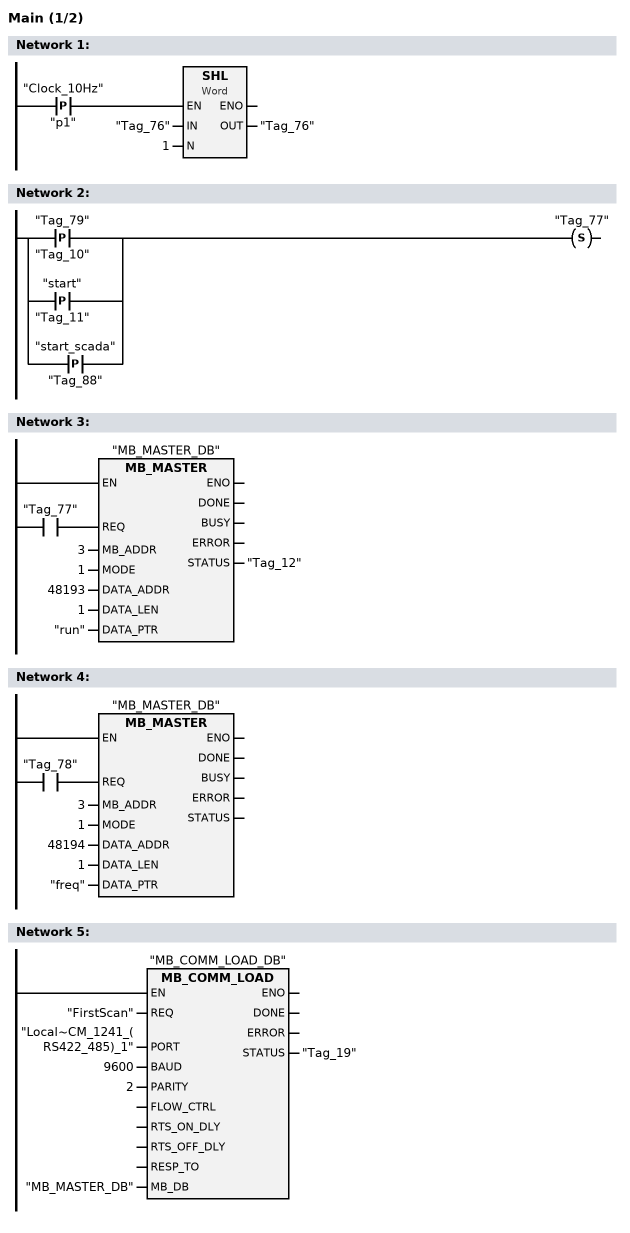
   RUNG wire#powerrail
      P_Contact(operand := "Clock_10Hz", bit := "p1")
      { S7_Templates := "SrcType := Word" } Shl(in := "Tag_76", n := 1, out => "Tag_76")
   END_RUNG
   // the same network as SCL:
   #_w1 := "Clock_10Hz" AND NOT "p1";   // rising edge of "Clock_10Hz"
   "p1" := "Clock_10Hz";
   IF #_w1 THEN "Tag_76" := SHL(IN := "Tag_76", N := 1); END_IF;
END_REGION

REGION Network 2
   RUNG wire#powerrail
      P_Contact(operand := "Tag_79", bit := "Tag_10")
      wire#w1
      S_Coil( "Tag_77" )
   END_RUNG
   RUNG wire#powerrail
      P_Contact(operand := "start", bit := "Tag_11")
   END_RUNG wire#w1
   RUNG wire#powerrail
      P_Contact(operand := "start_scada", bit := "Tag_88")
   END_RUNG wire#w1
   // the same network as SCL:
   #_w1 := "Tag_79" AND NOT "Tag_10";   // rising edge of "Tag_79"
   "Tag_10" := "Tag_79";
   #_w2 := "start" AND NOT "Tag_11";   // rising edge of "start"
   "Tag_11" := "start";
   #_w3 := "start_scada" AND NOT "Tag_88";   // rising edge of "start_scada"
   "Tag_88" := "start_scada";
   IF #_w1 OR #_w2 OR #_w3 THEN "Tag_77" := TRUE; END_IF;
END_REGION

REGION Network 3
   "MB_MASTER_DB"(REQ := "Tag_77",   // MB_MASTER
                  MB_ADDR := 3,
                  MODE := 1,
                  DATA_ADDR := 48193,
                  DATA_LEN := 1,
                  DATA_PTR := "run",
                  STATUS => "Tag_12");
END_REGION

REGION Network 4
   "MB_MASTER_DB"(REQ := "Tag_78",   // MB_MASTER
                  MB_ADDR := 3,
                  MODE := 1,
                  DATA_ADDR := 48194,
                  DATA_LEN := 1,
                  DATA_PTR := "freq");
END_REGION

REGION Network 5
   "MB_COMM_LOAD_DB"(REQ := "FirstScan",   // MB_COMM_LOAD
                     PORT := "Local~CM_1241_(RS422_485)_1",
                     BAUD := 9600,
                     PARITY := 2,
                     MB_DB := "MB_MASTER_DB",
                     STATUS => "Tag_19");
END_REGION

REGION Network 6
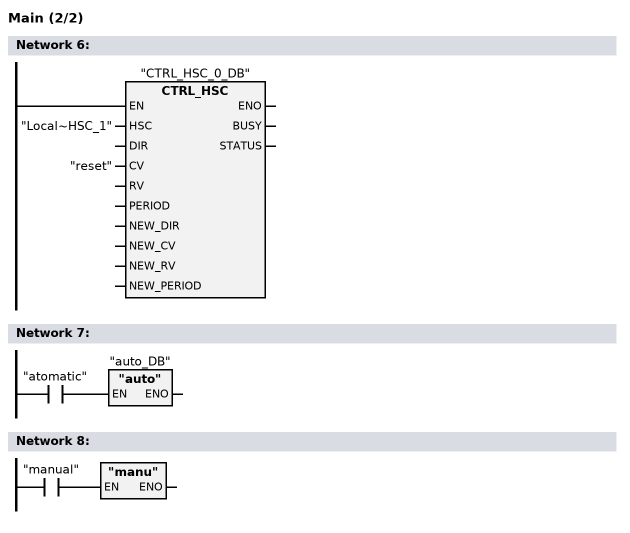
   "CTRL_HSC_0_DB"(HSC := "Local~HSC_1", CV := "reset");   // CTRL_HSC
END_REGION

REGION Network 7
   RUNG wire#powerrail
      Contact( "atomatic" )
      "auto_DB"()
   END_RUNG
   // the same network as SCL:
   IF "atomatic" THEN
       "auto_DB"();   // "auto"
   END_IF;
END_REGION

REGION Network 8
   RUNG wire#powerrail
      Contact( "manual" )
      "manu"()
   END_RUNG
   // the same network as SCL:
   IF "manual" THEN "manu"(); END_IF;
END_REGION
END_ORGANIZATION_BLOCK

// ===== PLC "PLC_3"  CPU 1212C AC/DC/Rly =====

VAR_GLOBAL   // PLC tag table "Default tag table"
   "Tag_1" AT %M3.1 : Bool;
   "Tag_2" AT %M3.2 : Bool;
   "Tag_3" AT %M3.3 : Bool;
   "Tag_4" AT %M3.4 : Bool;
   "Tag_5" AT %M0.0 : Bool;
   "Tag_6" AT %MW2 : Word;
   "Tag_7" AT %MW10 : Word;
   "Tag_8" AT %MW12 : Word;
   "Tag_9" AT %M150.0 : Bool;
END_VAR

ORGANIZATION_BLOCK "Main"   // OB1, LAD, ProgramCycle
TITLE = "Main Program Sweep (Cycle)"
{ S7_Optimized_Access := 'TRUE' }
VERSION : 0.1
BEGIN

REGION Network 2
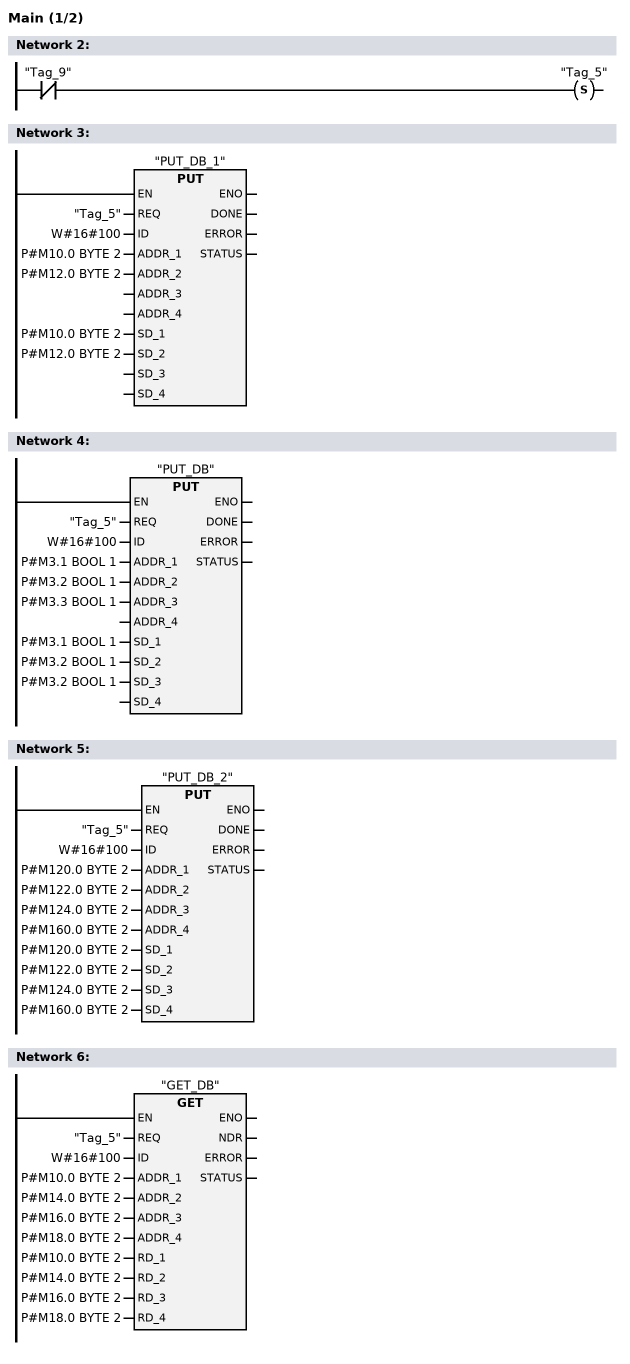
   RUNG wire#powerrail
      I_Contact( "Tag_9" )
      S_Coil( "Tag_5" )
   END_RUNG
   // the same network as SCL:
   IF NOT "Tag_9" THEN "Tag_5" := TRUE; END_IF;
END_REGION

REGION Network 3
   "PUT_DB_1"(REQ := "Tag_5",   // PUT
              ID := W#16#100,
              ADDR_1 := P#M10.0 BYTE 2,
              ADDR_2 := P#M12.0 BYTE 2,
              SD_1 := P#M10.0 BYTE 2,
              SD_2 := P#M12.0 BYTE 2);
END_REGION

REGION Network 4
   "PUT_DB"(REQ := "Tag_5",   // PUT
            ID := W#16#100,
            ADDR_1 := P#M3.1 BOOL 1,
            ADDR_2 := P#M3.2 BOOL 1,
            ADDR_3 := P#M3.3 BOOL 1,
            SD_1 := P#M3.1 BOOL 1,
            SD_2 := P#M3.2 BOOL 1,
            SD_3 := P#M3.2 BOOL 1);
END_REGION

REGION Network 5
   "PUT_DB_2"(REQ := "Tag_5",   // PUT
              ID := W#16#100,
              ADDR_1 := P#M120.0 BYTE 2,
              ADDR_2 := P#M122.0 BYTE 2,
              ADDR_3 := P#M124.0 BYTE 2,
              ADDR_4 := P#M160.0 BYTE 2,
              SD_1 := P#M120.0 BYTE 2,
              SD_2 := P#M122.0 BYTE 2,
              SD_3 := P#M124.0 BYTE 2,
              SD_4 := P#M160.0 BYTE 2);
END_REGION

REGION Network 6
   "GET_DB"(REQ := "Tag_5",   // GET
            ID := W#16#100,
            ADDR_1 := P#M10.0 BYTE 2,
            ADDR_2 := P#M14.0 BYTE 2,
            ADDR_3 := P#M16.0 BYTE 2,
            ADDR_4 := P#M18.0 BYTE 2,
            RD_1 := P#M10.0 BYTE 2,
            RD_2 := P#M14.0 BYTE 2,
            RD_3 := P#M16.0 BYTE 2,
            RD_4 := P#M18.0 BYTE 2);
END_REGION

REGION Network 8
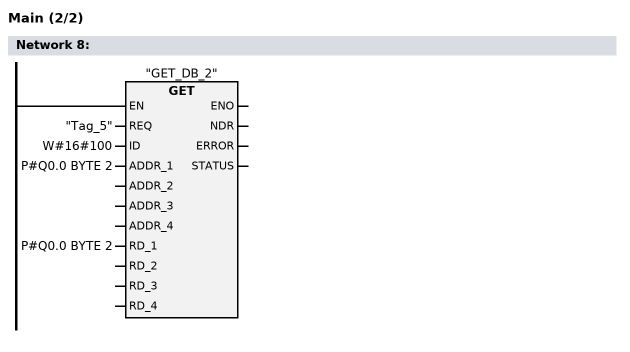
   "GET_DB_2"(REQ := "Tag_5", ID := W#16#100, ADDR_1 := P#Q0.0 BYTE 2, RD_1 := P#Q0.0 BYTE 2);   // GET
END_REGION
END_ORGANIZATION_BLOCK